// TIA Portal V20 export
// export: Created 2026-07-10T11:12:33.3603601Z, ExportSetting WithDefaults, DisplayName Totally Integrated Automation Portal, DisplayVersion V20, DisplayName TIA Portal Openness, DisplayVersion V20, DisplayName TIA Portal Version Control Interface, DisplayVersion V20, DisplayName STEP 7 Professional, DisplayVersion V20, DisplayName STEP 7 Safety, DisplayVersion V20, DisplayName WinCC Basic/Comfort/Advanced, DisplayVersion V20, DisplayName WinCC Unified, DisplayVersion V20
FUNCTION_BLOCK "MotorControllerSimple"   // FB12, SCL
{ S7_Optimized_Access := 'TRUE' }
VERSION : 0.1
// stored: AutoNumber true, IsIECCheckEnabled false, IsRetainMemResEnabled false, MemoryReserve 100, SetENOAutomatically false, UDAEnableTagReadback false
   VAR_INPUT
      Enable : Bool;
      CurrentPosition : Real;
      SetpointPosition : Real;
      PositionDeadzone : Real := 2.0;
      MinimalPulse : Time;
      PauseMode : Time := T#10s;
      isMoving : Bool;
      MoveNow : Bool;
      MinReversPause : Time := T#1s;
      PositionError : Bool;
   END_VAR
   VAR_OUTPUT
      Open : Bool;
      Close : Bool;
   END_VAR
   VAR
      Opening : Bool;
      Closing : Bool;
      MovingTOF { S7_SetPoint := 'True'} : TOF_TIME;
      OpeningTOF { S7_SetPoint := 'True'} : TOF_TIME;
      ClosingTOF { S7_SetPoint := 'True'} : TOF_TIME;
      TON1 { S7_SetPoint := 'True'} : TON_TIME;
      TON2 { S7_SetPoint := 'True'} : TON_TIME;
   END_VAR
BEGIN
   #MovingTOF(IN:=(#isMoving OR #Open OR #Close),
              PT:=#PauseMode);
   #OpeningTOF(IN:=#Open,
               PT:=#MinReversPause);
   #ClosingTOF(IN:=#Close,
               PT:=#MinReversPause);

   IF #Enable AND NOT #PositionError THEN
       IF (NOT #MovingTOF.Q) OR #MoveNow THEN
           IF #CurrentPosition < #SetpointPosition - #PositionDeadzone THEN
               #Opening := TRUE;
               #Closing := FALSE;
           END_IF;
           IF #CurrentPosition > #SetpointPosition + #PositionDeadzone THEN
               #Opening := FALSE;
               #Closing := TRUE;
           END_IF;
           IF #SetpointPosition = 0 THEN
               #Opening := FALSE;
               #Closing := TRUE;
           END_IF;
           IF #SetpointPosition = 100 THEN
               #Opening := TRUE;
               #Closing := FALSE;
           END_IF;

       END_IF;

       IF #Opening AND #CurrentPosition >= #SetpointPosition - 0.1 THEN
           #Opening := FALSE;
       END_IF;
       IF #Closing AND #CurrentPosition <= #SetpointPosition + 0.1 THEN
           #Closing := FALSE;
       END_IF;

       IF #Opening AND (NOT #ClosingTOF.Q) THEN
           #Open := TRUE;
       ELSIF (NOT #Opening) AND #TON1.Q THEN
           #Open := FALSE;
       END_IF;

       #TON1(IN:=#Open,
             PT:=#MinimalPulse);

       IF #Closing AND (NOT #OpeningTOF.Q) THEN
           #Close := TRUE;
       ELSIF (NOT #Closing) AND #TON2.Q THEN
           #Close := FALSE;
       END_IF;

       #TON2(IN:=#Close,
             PT:=#MinimalPulse);
   ELSE
       #Open := FALSE;
       #Close := FALSE;
       #Opening := FALSE;
       #Closing := FALSE;
       RESET_TIMER(#TON1);
       RESET_TIMER(#TON2);
   END_IF;
END_FUNCTION_BLOCK
